TYPE ST_System_DLK_Parameter :
STRUCT
	AutoQuittierung			: BOOL;

END_STRUCT
END_TYPE

(* stored: Version 1.1.0.1, ProductVersion 3.1.4024.9
   DUT ST_System_DLK_Parameter: Id {86ff32c4-bd69-475d-9749-ab38d70e25e6} *)
